// Tests for AstroBROT.FB_HADEC2RADEC (apparent hour angle / Dec -> ICRS RA/Dec; the block IAG50cm uses).
//
// GENERATED by AstroBROT/testing/gen_block_tests.py from testing/golden_blocks.py, do not edit the numbers by hand.
// Every golden case is checked against the Python port of the ST (1E-7 deg) and against erfa.atoc13 as a great-circle
// separation on the sky (2E-4 deg = 0.72 arcsec).
//
// KNOWN LIMITATION, pinned here on purpose: at exactly dec = +-90 the ST applies the aberration and nutation
// corrections in (ra, dec), d_ra grows like 1/cos(dec) and the dec correction is evaluated at an RA that means
// nothing there. The result then depends on the hour angle and is 4.7 arcsec (north) / 39 arcsec (south) away from
// erfa. Golden_Exact_Poles allows 0.015 deg so that it cannot get worse unnoticed; 0.1 deg from the pole the error is
// back at 0.5 arcsec (Golden_Near_The_Poles, strict tolerance).
FUNCTION_BLOCK FB_HADEC2RADEC_Tests EXTENDS TcUnit.FB_TestSuite
VAR
END_VAR

Golden_Tenerife_2026();
Golden_Tenerife_low();
Golden_South_2010();
Golden_Dut1();
Golden_HA_Wrap();
Golden_Near_The_Poles();
Golden_Exact_Poles();
Hour_Angle_Is_Periodic();
Longitude_Is_Periodic();
Outputs_Stay_In_Range();
Round_Trip_Through_RADEC2HADEC();
Inputs_Are_Not_Modified();
Cyclic_Calls_With_Inputs_Set_Once_Are_Stable();

METHOD PRIVATE CheckNear
VAR_INPUT
	fExpected	: LREAL;
	fActual	: LREAL;
	fDelta	: LREAL;
	sName	: STRING(255);
END_VAR
AssertEquals_LREAL(Expected := fExpected, Actual := fActual, Delta := fDelta, Message := sName);
END_METHOD

METHOD PRIVATE CheckAngle
VAR_INPUT
	fExpected	: LREAL;
	fActual	: LREAL;
	fDelta	: LREAL;
	sName	: STRING(255);
END_VAR
VAR
	fDiff	: LREAL;
END_VAR
// angles in degrees, compared modulo 360 so that 359.9999999 and -1.0E-7 are equal
fDiff := fActual - fExpected;
WHILE fDiff > 180.0 DO fDiff := fDiff - 360.0; END_WHILE
WHILE fDiff < -180.0 DO fDiff := fDiff + 360.0; END_WHILE
AssertEquals_LREAL(Expected := 0.0, Actual := fDiff, Delta := fDelta, Message := sName);
END_METHOD

METHOD PRIVATE CheckSeparation
VAR_INPUT
	fLon1	: LREAL;
	fLat1	: LREAL;
	fLon2	: LREAL;
	fLat2	: LREAL;
	fDelta	: LREAL;
	sName	: STRING(255);
END_VAR
VAR
	fD2r	: LREAL;
	fHalfDLat	: LREAL;
	fHalfDLon	: LREAL;
	fHav	: LREAL;
	fSep	: LREAL;
END_VAR
// great-circle separation of two positions (longitude, latitude in degrees) against a tolerance in degrees;
// a difference of longitudes is not a distance on the sky, this is (haversine formula)
fD2r := 0.017453292519943295;
fHalfDLat := (fLat2 - fLat1) * fD2r * 0.5;
fHalfDLon := (fLon2 - fLon1) * fD2r * 0.5;
fHav := SIN(fHalfDLat) * SIN(fHalfDLat) + COS(fLat1 * fD2r) * COS(fLat2 * fD2r) * SIN(fHalfDLon) * SIN(fHalfDLon);
fSep := 2.0 * ASIN(SQRT(LIMIT(0.0, fHav, 1.0))) / fD2r;
AssertEquals_LREAL(Expected := 0.0, Actual := fSep, Delta := fDelta, Message := sName);
END_METHOD

METHOD PRIVATE Golden_Tenerife_2026
VAR
	fb	: AstroBROT.FB_HADEC2RADEC;
END_VAR
TEST('Golden_Tenerife_2026');
fb(jd := 2461300.75, ha := 345.0, dec := 22.01, lon := -16.5, dut1 := 0.0);
CheckAngle(84.28759958479777, fb.ra_out, 1.0E-7, 'Tenerife_2026 ra');
CheckNear(21.993212482320583, fb.dec_out, 1.0E-7, 'Tenerife_2026 dec');
CheckSeparation(84.28749809589803, 21.9932192971722, fb.ra_out, fb.dec_out, 0.0002, 'Tenerife_2026 vs erfa');
TEST_FINISHED();
END_METHOD

METHOD PRIVATE Golden_Tenerife_low
VAR
	fb	: AstroBROT.FB_HADEC2RADEC;
END_VAR
TEST('Golden_Tenerife_low');
fb(jd := 2461300.75, ha := 30.0, dec := -10.0, lon := -16.5, dut1 := 0.0);
CheckAngle(39.36056226713681, fb.ra_out, 1.0E-7, 'Tenerife_low ra');
CheckNear(-10.11975028485237, fb.dec_out, 1.0E-7, 'Tenerife_low dec');
CheckSeparation(39.36047119642502, -10.11974494836338, fb.ra_out, fb.dec_out, 0.0002, 'Tenerife_low vs erfa');
TEST_FINISHED();
END_METHOD

METHOD PRIVATE Golden_South_2010
VAR
	fb	: AstroBROT.FB_HADEC2RADEC;
END_VAR
TEST('Golden_South_2010');
fb(jd := 2455197.5, ha := 100.0, dec := -47.3, lon := -70.7, dut1 := 0.0);
CheckAngle(289.6589544745373, fb.ra_out, 1.0E-7, 'South_2010 ra');
CheckNear(-47.317658585279744, fb.dec_out, 1.0E-7, 'South_2010 dec');
CheckSeparation(289.65896142189746, -47.31759859445048, fb.ra_out, fb.dec_out, 0.0002, 'South_2010 vs erfa');
TEST_FINISHED();
END_METHOD

METHOD PRIVATE Golden_Dut1
VAR
	fb	: AstroBROT.FB_HADEC2RADEC;
END_VAR
TEST('Golden_Dut1');
fb(jd := 2461300.75, ha := 345.0, dec := 22.01, lon := -16.5, dut1 := 0.9);
CheckAngle(84.29135982739001, fb.ra_out, 1.0E-7, 'Tenerife_dut1_plus ra');
CheckNear(21.993222245664892, fb.dec_out, 1.0E-7, 'Tenerife_dut1_plus dec');
CheckSeparation(84.2912582746304, 21.993229060334635, fb.ra_out, fb.dec_out, 0.0002, 'Tenerife_dut1_plus vs erfa');
fb(jd := 2461300.75, ha := 345.0, dec := 22.01, lon := -16.5, dut1 := -0.9);
CheckAngle(84.28383934246425, fb.ra_out, 1.0E-7, 'Tenerife_dut1_minus ra');
CheckNear(21.993202719039957, fb.dec_out, 1.0E-7, 'Tenerife_dut1_minus dec');
CheckSeparation(84.28373791742105, 21.993209534073422, fb.ra_out, fb.dec_out, 0.0002, 'Tenerife_dut1_minus vs erfa');
TEST_FINISHED();
END_METHOD

METHOD PRIVATE Golden_HA_Wrap
VAR
	fb	: AstroBROT.FB_HADEC2RADEC;
END_VAR
TEST('Golden_HA_Wrap');
fb(jd := 2461300.75, ha := 0.0001, dec := 22.01, lon := -16.5, dut1 := 0.0);
CheckAngle(69.28989220623771, fb.ra_out, 1.0E-7, 'HA_wrap_low ra');
CheckNear(21.955213314004528, fb.dec_out, 1.0E-7, 'HA_wrap_low dec');
CheckSeparation(69.28978714407457, 21.95521257782602, fb.ra_out, fb.dec_out, 0.0002, 'HA_wrap_low vs erfa');
fb(jd := 2461300.75, ha := 359.9999, dec := 22.01, lon := -16.5, dut1 := 0.0);
CheckAngle(69.29009214752863, fb.ra_out, 1.0E-7, 'HA_wrap_high ra');
CheckNear(21.95521380223834, fb.dec_out, 1.0E-7, 'HA_wrap_high dec');
CheckSeparation(69.28998708537415, 21.955213066161644, fb.ra_out, fb.dec_out, 0.0002, 'HA_wrap_high vs erfa');
TEST_FINISHED();
END_METHOD

METHOD PRIVATE Golden_Near_The_Poles
VAR
	fb	: AstroBROT.FB_HADEC2RADEC;
END_VAR
TEST('Golden_Near_The_Poles');
fb(jd := 2461300.75, ha := 200.0, dec := 89.9, lon := -16.5, dut1 := 0.0);
CheckAngle(316.7079065490832, fb.ra_out, 1.0E-7, 'Near_north_pole ra');
CheckNear(89.8844737036994, fb.dec_out, 1.0E-7, 'Near_north_pole dec');
CheckSeparation(316.7064081660361, 89.88445978947462, fb.ra_out, fb.dec_out, 0.0002, 'Near_north_pole vs erfa');
fb(jd := 2455197.5, ha := 200.0, dec := -89.9, lon := -70.7, dut1 := 0.0);
CheckAngle(186.30600937346122, fb.ra_out, 1.0E-7, 'Near_south_pole ra');
CheckNear(-89.84872530394176, fb.dec_out, 1.0E-7, 'Near_south_pole dec');
CheckSeparation(186.3367115207879, -89.84875262097749, fb.ra_out, fb.dec_out, 0.0002, 'Near_south_pole vs erfa');
TEST_FINISHED();
END_METHOD

METHOD PRIVATE Golden_Exact_Poles
VAR
	fb	: AstroBROT.FB_HADEC2RADEC;
END_VAR
TEST('Golden_Exact_Poles');
fb(jd := 2461300.75, ha := 200.0, dec := 90.0, lon := -16.5, dut1 := 0.0);
// at exactly dec = +-90 neither ra nor dec is reproducible (d_ra ~ 1/cos(dec) = 1E16, and d_dec is evaluated at that ra), only the bound against erfa is pinned
CheckSeparation(358.71048545509177, 89.85071696591022, fb.ra_out, fb.dec_out, 0.015, 'North_pole vs erfa');
fb(jd := 2455197.5, ha := 200.0, dec := -90.0, lon := -70.7, dut1 := 0.0);
// at exactly dec = +-90 neither ra nor dec is reproducible (d_ra ~ 1/cos(dec) = 1E16, and d_dec is evaluated at that ra), only the bound against erfa is pinned
CheckSeparation(179.80951066897055, -89.94824466951559, fb.ra_out, fb.dec_out, 0.015, 'South_pole vs erfa');
TEST_FINISHED();
END_METHOD

METHOD PRIVATE Hour_Angle_Is_Periodic
VAR
	fb	: AstroBROT.FB_HADEC2RADEC;
END_VAR
TEST('Hour_Angle_Is_Periodic');
// ha and ha +- 360 are the same position; the block does not wrap ra before the corrections, so this also covers the wrap of d_ra (issue #10)
fb(jd := 2461300.75, ha := -15.0, dec := 22.01, lon := -16.5);
CheckAngle(84.28759958479777, fb.ra_out, 1.0E-9, 'ha - 360 ra');
CheckNear(21.993212482320583, fb.dec_out, 1.0E-9, 'ha - 360 dec');
fb(jd := 2461300.75, ha := 705.0, dec := 22.01, lon := -16.5);
CheckAngle(84.28759958479777, fb.ra_out, 1.0E-9, 'ha + 360 ra');
CheckNear(21.993212482320583, fb.dec_out, 1.0E-9, 'ha + 360 dec');
AssertTrue(Condition := fb.ra_out >= 0.0 AND fb.ra_out < 360.0, Message := 'ra_out is within 0 <= ra < 360');
TEST_FINISHED();
END_METHOD

METHOD PRIVATE Longitude_Is_Periodic
VAR
	fb	: AstroBROT.FB_HADEC2RADEC;
END_VAR
TEST('Longitude_Is_Periodic');
fb(jd := 2461300.75, ha := 345.0, dec := 22.01, lon := 343.5);
CheckAngle(84.28759958479777, fb.ra_out, 1.0E-9, 'lon + 360 ra');
fb(jd := 2461300.75, ha := 345.0, dec := 22.01, lon := -376.5);
CheckAngle(84.28759958479777, fb.ra_out, 1.0E-9, 'lon - 360 ra');
TEST_FINISHED();
END_METHOD

METHOD PRIVATE Outputs_Stay_In_Range
VAR
	fb	: AstroBROT.FB_HADEC2RADEC;
	i	: INT;
	fHa	: LREAL;
END_VAR
TEST('Outputs_Stay_In_Range');
FOR i := -1 TO 8 DO
	fHa := 45.0 * i;
	fb(jd := 2461300.75, ha := fHa, dec := 89.9, lon := -16.5);
	AssertTrue(Condition := fb.ra_out >= 0.0 AND fb.ra_out < 360.0 AND fb.dec_out <= 90.0 AND fb.dec_out >= -90.0, Message := 'ha sweep at dec +89.9 stays in range');
	fb(jd := 2461300.75, ha := fHa, dec := -89.9, lon := -16.5);
	AssertTrue(Condition := fb.ra_out >= 0.0 AND fb.ra_out < 360.0 AND fb.dec_out <= 90.0 AND fb.dec_out >= -90.0, Message := 'ha sweep at dec -89.9 stays in range');
	fb(jd := 2461300.75, ha := fHa, dec := 0.0, lon := -16.5);
	AssertTrue(Condition := fb.ra_out >= 0.0 AND fb.ra_out < 360.0 AND fb.dec_out <= 90.0 AND fb.dec_out >= -90.0, Message := 'ha sweep at dec 0 stays in range');
END_FOR
TEST_FINISHED();
END_METHOD

METHOD PRIVATE Round_Trip_Through_RADEC2HADEC
VAR
	fbFwd	: AstroBROT.FB_RADEC2HADEC;
	fbBack	: AstroBROT.FB_HADEC2RADEC;
END_VAR
TEST('Round_Trip_Through_RADEC2HADEC');
// the two blocks are only approximate inverses (nutation and aberration are applied at slightly different
// positions), so 1E-6 deg away from the poles and 2E-4 deg (0.72 arcsec) 0.1 deg from a pole
fbFwd(jd := 2461300.75, ra := 83.63, dec := 22.01, lon := -16.5);
fbBack(jd := 2461300.75, ha := fbFwd.ha_out, dec := fbFwd.dec_out, lon := -16.5);
CheckSeparation(83.63, 22.01, fbBack.ra_out, fbBack.dec_out, 1.0E-6, 'Tenerife_2026');
fbFwd(jd := 2455197.5, ra := 312.5, dec := -47.3, lon := -70.7);
fbBack(jd := 2455197.5, ha := fbFwd.ha_out, dec := fbFwd.dec_out, lon := -70.7);
CheckSeparation(312.5, -47.3, fbBack.ra_out, fbBack.dec_out, 1.0E-6, 'South_2010');
fbFwd(jd := 2461300.75, ra := 359.9999, dec := 22.01, lon := -16.5);
fbBack(jd := 2461300.75, ha := fbFwd.ha_out, dec := fbFwd.dec_out, lon := -16.5);
CheckSeparation(359.9999, 22.01, fbBack.ra_out, fbBack.dec_out, 1.0E-6, 'RA just below 360');
fbFwd(jd := 2461300.75, ra := 0.0001, dec := 22.01, lon := -16.5);
fbBack(jd := 2461300.75, ha := fbFwd.ha_out, dec := fbFwd.dec_out, lon := -16.5);
CheckSeparation(0.0001, 22.01, fbBack.ra_out, fbBack.dec_out, 1.0E-6, 'RA just above 0');
fbFwd(jd := 2461300.75, ra := 200.0, dec := 89.9, lon := -16.5);
fbBack(jd := 2461300.75, ha := fbFwd.ha_out, dec := fbFwd.dec_out, lon := -16.5);
CheckSeparation(200.0, 89.9, fbBack.ra_out, fbBack.dec_out, 0.0002, 'near the north pole');
TEST_FINISHED();
END_METHOD

METHOD PRIVATE Inputs_Are_Not_Modified
VAR
	fb	: AstroBROT.FB_HADEC2RADEC;
END_VAR
TEST('Inputs_Are_Not_Modified');
fb(jd := 2461300.75, ha := 345.0, dec := 22.01, lon := -16.5, dut1 := 0.5);
CheckNear(2461300.75, fb.jd, 0.0, 'jd unchanged');
CheckNear(345.0, fb.ha, 0.0, 'ha unchanged');
CheckNear(22.01, fb.dec, 0.0, 'dec unchanged');
CheckNear(-16.5, fb.lon, 0.0, 'lon unchanged');
CheckNear(0.5, fb.dut1, 0.0, 'dut1 unchanged');
TEST_FINISHED();
END_METHOD

METHOD PRIVATE Cyclic_Calls_With_Inputs_Set_Once_Are_Stable
VAR
	fb	: AstroBROT.FB_HADEC2RADEC;
	i	: INT;
END_VAR
TEST('Cyclic_Calls_With_Inputs_Set_Once_Are_Stable');
fb.jd := 2461300.75;
fb.ha := 345.0;
fb.dec := 22.01;
fb.lon := -16.5;
FOR i := 1 TO 5 DO
	fb();
	CheckAngle(84.28759958479777, fb.ra_out, 1.0E-7, 'cyclic call ra');
	CheckNear(21.993212482320583, fb.dec_out, 1.0E-7, 'cyclic call dec');
END_FOR
TEST_FINISHED();
END_METHOD

END_FUNCTION_BLOCK

(* stored: Version 1.1.0.1, ProductVersion 3.1.4024.15
   POU FB_HADEC2RADEC_Tests: Id {3526ec90-a2e1-5bd2-8923-88726d720c9a}, SpecialFunc None
   Method CheckNear: Id {3803b234-6a4a-5f3e-ae8f-9be8ad93f31d}
   Method CheckAngle: Id {9dce2086-0c26-5a9b-ac55-9a52793bf4dd}
   Method CheckSeparation: Id {d3fde661-d6e5-5396-8e1b-a8b26fb7abaf}
   Method Golden_Tenerife_2026: Id {fa753f6d-8c99-5f36-913f-33469afcddc9}
   Method Golden_Tenerife_low: Id {5709d20d-fb31-5ef5-b8de-d304b995132a}
   Method Golden_South_2010: Id {60438eb9-7dde-5731-aac7-6f079c1d82a5}
   Method Golden_Dut1: Id {21636bce-a3f5-55c3-a93b-997d29707cf8}
   Method Golden_HA_Wrap: Id {b77b9d2b-bb62-50cc-a7d0-4744754e5056}
   Method Golden_Near_The_Poles: Id {b8533e73-d348-59d1-81c1-e5299d6e1d1c}
   Method Golden_Exact_Poles: Id {ed7ba411-c41c-5e83-b644-ac35d6995366}
   Method Hour_Angle_Is_Periodic: Id {6b513f48-ffc4-51ef-b615-38ae7ade21f3}
   Method Longitude_Is_Periodic: Id {0847667b-b68c-57b4-8bc1-ba794e99dcb4}
   Method Outputs_Stay_In_Range: Id {a8091054-9d20-565d-957d-3b81986f2485}
   Method Round_Trip_Through_RADEC2HADEC: Id {e58622d7-be22-5cc5-9f05-d2a3183d87a3}
   Method Inputs_Are_Not_Modified: Id {da5f922f-32bf-578b-b880-d28443b770be}
   Method Cyclic_Calls_With_Inputs_Set_Once_Are_Stable: Id {894e2f06-00a0-5f17-a4f7-92369f0c7a4a} *)
